// TIA Portal V20 export
TYPE "UDT_Alarms"
   STRUCT
      Id : DInt;
      Severity : Byte;
      Acknowledge : Bool;
   END_STRUCT;
END_TYPE
